INTERFACE I_AI_Voltage

PROPERTY errId : HAL_ErrorEnum
GET
END_GET
END_PROPERTY

PROPERTY rValue : real
GET
END_GET
END_PROPERTY

END_INTERFACE

(* stored: Version 1.1.0.1, ProductVersion 3.1.4024.6
   Itf I_AI_Voltage: Id {c02f3bf2-d011-0cf8-00c6-b63f55ae0d1f}
   Property errId: Id {1bd7bf6d-928b-064d-1547-c581aa92035d}
   Get Get: Id {5b6596ce-6480-0062-1771-ed368dc30ae1}
   Property rValue: Id {dd1fe455-e7ca-0b34-3bfb-13e702cf2e53}
   Get Get: Id {23242fee-e46a-0a70-1022-0006b5897ed1} *)
